{attribute 'qualified_only'}
VAR_GLOBAL
	HWIO		:HardWareIO;
END_VAR

(* stored: Version 1.1.0.1, ProductVersion 3.1.4022.16
   GVL GVL_Machine: Id {c39f9a5e-bc46-47e8-9a07-5b407580079f} *)
